// Mitsubishi GX Works2 project: 04-06-2020 EX3   PLC: FX3U/FX3UC

PROGRAM MAIN
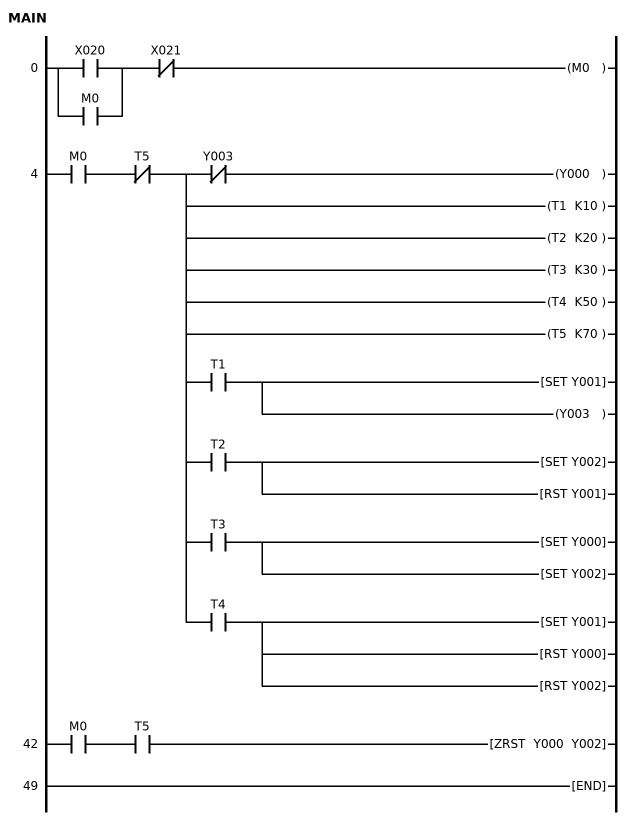
0     LD      X020
      OR      M0
      ANI     X021
      OUT     M0
4     LD      M0
      ANI     T5
      MPS
      ANI     Y003
      OUT     Y000
      MPP
      OUT     T1 K10
      OUT     T2 K20
      OUT     T3 K30
      OUT     T4 K50
      OUT     T5 K70
      MPS
      AND     T1
      SET     Y001
      OUT     Y003
      MRD
      AND     T2
      SET     Y002
      RST     Y001
      MRD
      AND     T3
      SET     Y000
      SET     Y002
      MPP
      AND     T4
      SET     Y001
      RST     Y000
      RST     Y002
42    LD      M0
      AND     T5
      ZRST    Y000 Y002
49    END
END_PROGRAM
